Fanuc TP program (LS listing): PNS0002.LS

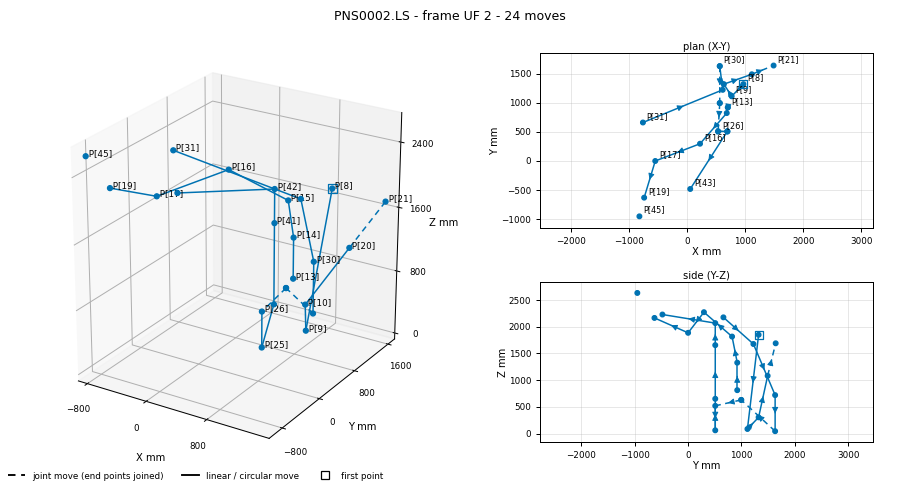
[picture p0: tool path of PNS0002.LS in frame UF 2, 24 of 53 moves have a stored position in this frame; points joined in program order, loops and branches not executed]
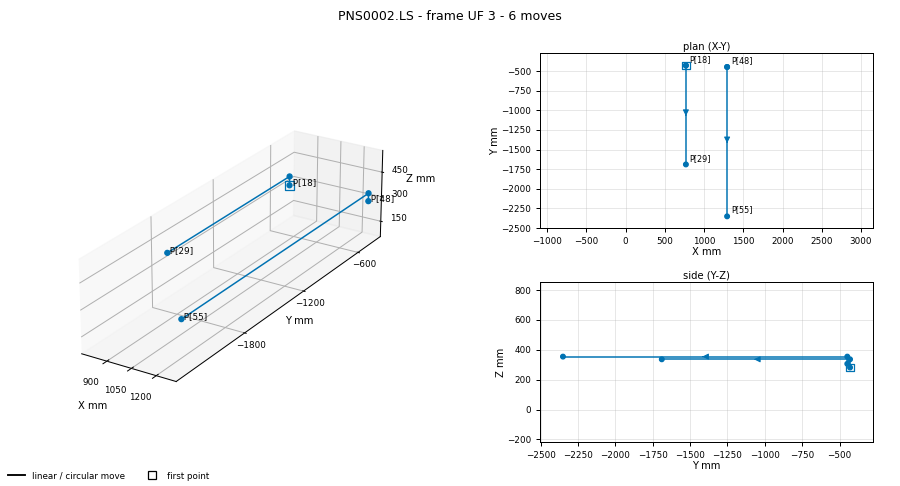
[picture p1: tool path of PNS0002.LS in frame UF 3, 6 of 53 moves have a stored position in this frame; points joined in program order, loops and branches not executed]
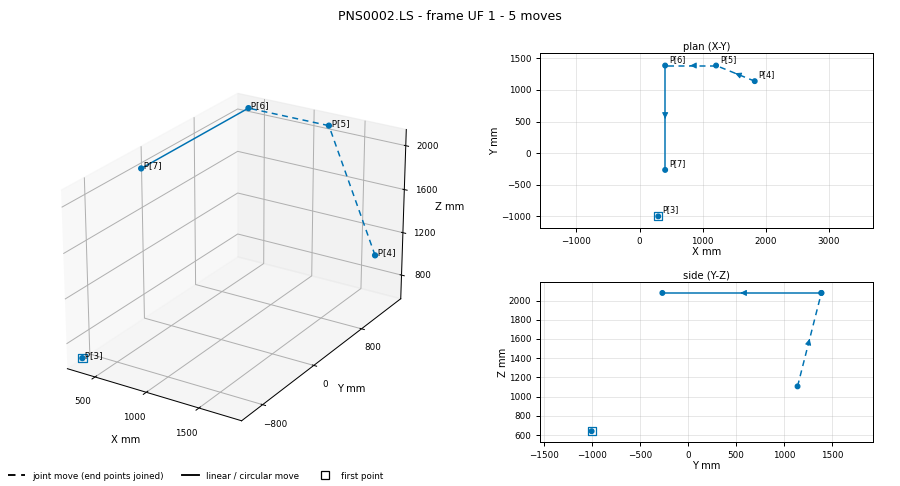
[picture p2: tool path of PNS0002.LS in frame UF 1, 5 of 53 moves have a stored position in this frame; points joined in program order, loops and branches not executed]
/PROG  PNS0002
/ATTR
OWNER		= MNEDITOR;
COMMENT		= "6410816256";
PROG_SIZE	= 5179;
CREATE		= DATE 26-03-31  TIME 11:21:30;
MODIFIED	= DATE 08-10-08  TIME 01:42:36;
FILE_NAME	= ;
VERSION		= 0;
LINE_COUNT	= 173;
MEMORY_SIZE	= 5531;
PROTECT		= READ_WRITE;
STORAGE		= CMOS;
TCD:  STACK_SIZE	= 0,
      TASK_PRIORITY	= 50,
      TIME_SLICE	= 0,
      BUSY_LAMP_OFF	= 0,
      ABORT_REQUEST	= 0,
      PAUSE_REQUEST	= 0;
DEFAULT_GROUP	= 1,*,*,*,*;
CONTROL_CODE	= 00000000 00000000;
/MN
   1:  !6410816256 ;
   2:  !--- INITIALIZE --- ;
   3:  UFRAME_NUM=0 ;
   4:  UTOOL_NUM=1 ;
   5:   ;
   6:J PR[1:HOME] 100% CNT50    ;
   7:   ;
   8:   ;
   9:   ;
  10:  !--- PICK --- ;
  11:  UFRAME_NUM=1 ;
  12:  UTOOL_NUM=1 ;
  13:  TIMER[1]=RESET ;
  14:  TIMER[1]=START ;
  15:   ;
  16:J P[3:INTMPT] 100% CNT10    ;
  17:L P[1:IN FRONT OF IF] 2000mm/sec CNT10    ;
  18:L P[2:ROTATE OVER PICK] 2000mm/sec CNT10    ;
  19:   ;
  20:  !INSERT PART PR ;
  21:  PR[2,3:OFFSET]=400    ;
  22:   ;
  23:L PR[51] 2000mm/sec FINE Offset,PR[2:OFFSET]    ;
  24:L PR[51] 700mm/sec FINE    ;
  25:   ;
  26:  CALL ALL_VAC_ON    ;
  27:   ;
  28:  WAIT   1.00(sec) ;
  29:   ;
  30:L PR[51] 700mm/sec FINE Offset,PR[2:OFFSET]    ;
  31:   ;
  32:J P[4:INTMPT] 100% CNT100    ;
  33:J P[5:INTMPT] 100% CNT100    ;
  34:J P[6:INTMPT] 100% CNT100    ;
  35:L P[7:INTMPT] 2000mm/sec CNT100    ;
  36:   ;
  37:  !--- ZERO TABLE --- ;
  38:  UFRAME_NUM=2 ;
  39:   ;
  40:L P[8:ABOVE ZERO] 1500mm/sec FINE    ;
  41:L P[9:ON ZERO] 1200mm/sec FINE    ;
  42:   ;
  43:  CALL ALL_VAC_OFF    ;
  44:   ;
  45:  !RE-PICK ;
  46:L P[10] 1500mm/sec FINE    ;
  47:L P[20] 1500mm/sec CNT100    ;
  48:J P[21:ROTATE 1] 75% CNT100    ;
  49:J P[22:ROTATE 2] 75% CNT100    ;
  50:J P[11] 75% CNT100    ;
  51:L P[12] 100mm/sec FINE    ;
  52:   ;
  53:  CALL ALL_VAC_ON    ;
  54:   ;
  55:  WAIT   1.00(sec) ;
  56:   ;
  57:L P[11] 155mm/sec FINE    ;
  58:   ;
  59:  !MOVE TO PRESS BREAK ;
  60:L P[13] 2000mm/sec CNT100    ;
  61:L P[14] 1500mm/sec CNT100    ;
  62:L P[15] 1500mm/sec CNT100    ;
  63:L P[16] 1500mm/sec CNT100    ;
  64:L P[17] 1500mm/sec CNT100    ;
  65:   ;
  66:L P[19:STAGED FOR BEND] 500mm/sec FINE    ;
  67:   ;
  68:  !--- BEND 1 --- ;
  69:  UFRAME_NUM=3 ;
  70:   ;
  71:L P[18:INSERT] 500mm/sec FINE    ;
  72:   ;
  73:  CALL PINCH    ;
  74:   ;
  75:  WAIT    .75(sec) ;
  76:   ;
  77:  CALL ALL_VAC_OFF    ;
  78:   ;
  79:  WAIT    .50(sec) ;
  80:   ;
  81:  CALL BEND    ;
  82:   ;
  83:  WAIT   1.00(sec) ;
  84:   ;
  85:  CALL ALL_VAC_ON    ;
  86:   ;
  87:  WAIT   1.00(sec) ;
  88:   ;
  89:  !OUT OF PRESS BREAK ;
  90:L P[28] 700mm/sec FINE    ;
  91:L P[29] 1200mm/sec CNT100    ;
  92:   ;
  93:  !--- ZERO TABLE --- ;
  94:  UFRAME_NUM=2 ;
  95:   ;
  96:  !MOVE TO ZERO ;
  97:L P[31] 1500mm/sec CNT100    ;
  98:L P[32] 1500mm/sec CNT100    ;
  99:L P[30] 1500mm/sec CNT100    ;
 100:L P[33] 500mm/sec FINE    ;
 101:   ;
 102:  CALL ALL_VAC_OFF    ;
 103:   ;
 104:  !REPOS FOR BEND 2 ;
 105:J P[23] 100% CNT100    ;
 106:   ;
 107:J P[24:ZERO J6] 100% CNT100    ;
 108:   ;
 109:J P[26] 100% CNT100    ;
 110:L P[25] 500mm/sec FINE    ;
 111:   ;
 112:L P[27] 1500mm/sec FINE    ;
 113:   ;
 114:  CALL ALL_VAC_ON    ;
 115:   ;
 116:  WAIT   1.00(sec) ;
 117:   ;
 118:  !MOVE TO PRESS BREAK ;
 119:L P[41] 500mm/sec CNT100    ;
 120:L P[42] 1200mm/sec CNT100    ;
 121:L P[43] 1200mm/sec CNT100    ;
 122:L P[44] 1200mm/sec CNT100    ;
 123:L P[45] 1500mm/sec CNT100    ;
 124:   ;
 125:  !--- BEND 2 --- ;
 126:  UFRAME_NUM=3 ;
 127:   ;
 128:L P[48] 500mm/sec FINE    ;
 129:   ;
 130:  CALL PINCH    ;
 131:   ;
 132:  WAIT    .75(sec) ;
 133:   ;
 134:  CALL ALL_VAC_OFF    ;
 135:   ;
 136:  WAIT    .50(sec) ;
 137:   ;
 138:  CALL BEND    ;
 139:   ;
 140:  WAIT   1.00(sec) ;
 141:   ;
 142:  CALL ALL_VAC_ON    ;
 143:   ;
 144:  WAIT   1.00(sec) ;
 145:   ;
 146:  !OUT OF INFEED ;
 147:L P[54] 500mm/sec CNT100    ;
 148:L P[55] 1200mm/sec CNT100    ;
 149:   ;
 150:  !--- OUTFEED --- ;
 151:  UFRAME_NUM=4 ;
 152:   ;
 153:L P[56] 1200mm/sec CNT100    ;
 154:L P[57] 1200mm/sec CNT100    ;
 155:L P[58] 1500mm/sec CNT100    ;
 156:L P[59] 1500mm/sec FINE Offset,PR[2:OFFSET]    ;
 157:L P[59] 500mm/sec FINE    ;
 158:   ;
 159:  CALL ALL_VAC_OFF    ;
 160:   ;
 161:L P[59] 1200mm/sec FINE Offset,PR[2:OFFSET]    ;
 162:   ;
 163:J PR[1:HOME] 100% CNT100    ;
 164:   ;
 165:  TIMER[1]=STOP ;
 166:  R[20]=(TIMER[1]) ;
 167:  !MOVE TO ZERO TABLE ;
 168:  !RE-PICK ;
 169:  !MOVE TO BREAK ;
 170:  !BREAK 1 ;
 171:  !BREAK 2 ;
 172:  !OUTFEED DROP ;
 173:  !HOME ;
/POS
P[1:"IN FRONT OF IF"]{
   GP1:
	UF : 0, UT : 1,		CONFIG : 'N U T, 0, 0, 0',
	X =  3074.267  mm,	Y =      .000  mm,	Z =  -312.592  mm,
	W =   180.000 deg,	P =     -.000 deg,	R =     -.000 deg,
	E1=  1548.896  mm
};
P[2:"ROTATE OVER PICK"]{
   GP1:
	UF : 0, UT : 1,		CONFIG : 'N U T, 0, 0, 0',
	X =  3074.267  mm,	Y =  1357.438  mm,	Z =  -312.592  mm,
	W =   180.000 deg,	P =      .000 deg,	R =    90.000 deg,
	E1=  2600.652  mm
};
P[3:"INTMPT"]{
   GP1:
	UF : 1, UT : 1,		CONFIG : 'N U T, 0, 0, 0',
	X =   295.983  mm,	Y = -1001.060  mm,	Z =   641.268  mm,
	W =   180.000 deg,	P =     -.000 deg,	R =     -.000 deg,
	E1=   633.339  mm
};
P[4:"INTMPT"]{
   GP1:
	UF : 1, UT : 1,		CONFIG : 'N U T, 0, 0, 0',
	X =  1823.555  mm,	Y =  1139.742  mm,	Z =  1107.202  mm,
	W =   180.000 deg,	P =   -40.393 deg,	R =    90.000 deg,
	E1=  2600.652  mm
};
P[5:"INTMPT"]{
   GP1:
	UF : 1, UT : 1,		CONFIG : 'N U T, 0, 0, 0',
	X =  1211.540  mm,	Y =  1387.428  mm,	Z =  2078.739  mm,
	W =   -90.000 deg,	P =   -90.000 deg,	R =     0.000 deg,
	E1=  2600.652  mm
};
P[6:"INTMPT"]{
   GP1:
	UF : 1, UT : 1,		CONFIG : 'N U T, 0, -1, 1',
	X =   405.131  mm,	Y =  1387.428  mm,	Z =  2078.739  mm,
	W =  -111.305 deg,	P =   -90.000 deg,	R =     0.000 deg,
	E1=  1672.415  mm
};
P[7:"INTMPT"]{
   GP1:
	UF : 1, UT : 1,		CONFIG : 'N U T, 0, -1, 1',
	X =   405.131  mm,	Y =  -265.705  mm,	Z =  2078.738  mm,
	W =  -162.943 deg,	P =   -90.000 deg,	R =     0.000 deg,
	E1=  1243.168  mm
};
P[8:"ABOVE ZERO"]{
   GP1:
	UF : 2, UT : 1,		CONFIG : 'N U T, 0, -1, 1',
	X =   970.105  mm,	Y =  1320.827  mm,	Z =  1850.509  mm,
	W =  -179.999 deg,	P =      .001 deg,	R =      .000 deg,
	E1=  2140.441  mm
};
P[9:"ON ZERO"]{
   GP1:
	UF : 2, UT : 1,		CONFIG : 'N U T, 0, -1, 1',
	X =   769.156  mm,	Y =  1111.796  mm,	Z =    85.489  mm,
	W =  -179.997 deg,	P =      .005 deg,	R =     -.999 deg,
	E1=  2580.816  mm
};
P[10:""]{
   GP1:
	UF : 2, UT : 1,		CONFIG : 'N U T, 0, -1, 1',
	X =   635.159  mm,	Y =  1320.793  mm,	Z =   303.508  mm,
	W =  -179.998 deg,	P =      .003 deg,	R =      .000 deg,
	E1=  2580.816  mm
};
P[11:""]{
   GP1:
	UF : 2, UT : 1,
	J1=    18.263 deg,	J2=     6.836 deg,	J3=    -5.826 deg,
	J4=    40.003 deg,	J5=   -26.642 deg,	J6=   234.609 deg,
	E1=  2580.816  mm
};
P[12:""]{
   GP1:
	UF : 2, UT : 1,
	J1=    15.187 deg,	J2=    25.137 deg,	J3=    -9.019 deg,
	J4=    39.754 deg,	J5=   -22.236 deg,	J6=   235.320 deg,
	E1=  2580.816  mm
};
P[13]{
   GP1:
	UF : 2, UT : 1,		CONFIG : 'N U T, 0, -1, 1',
	X =   702.535  mm,	Y =   920.780  mm,	Z =   812.300  mm,
	W =  -179.997 deg,	P =      .004 deg,	R =      .000 deg,
	E1=  2580.816  mm
};
P[14]{
   GP1:
	UF : 2, UT : 1,		CONFIG : 'N U T, 0, 0, 0',
	X =   702.534  mm,	Y =   920.780  mm,	Z =  1327.631  mm,
	W =  -179.997 deg,	P =      .004 deg,	R =      .000 deg,
	E1=  2221.229  mm
};
P[15]{
   GP1:
	UF : 2, UT : 1,		CONFIG : 'N U T, 0, 0, 0',
	X =   684.474  mm,	Y =   823.810  mm,	Z =  1816.677  mm,
	W =   151.491 deg,	P =      .004 deg,	R =     -.001 deg,
	E1=  2195.893  mm
};
P[16]{
   GP1:
	UF : 2, UT : 1,		CONFIG : 'N U T, 0, 0, 1',
	X =   225.090  mm,	Y =   296.601  mm,	Z =  2273.432  mm,
	W =   117.226 deg,	P =    -8.632 deg,	R =   -56.480 deg,
	E1=  1531.414  mm
};
P[17]{
   GP1:
	UF : 2, UT : 1,		CONFIG : 'N U T, 0, 0, 1',
	X =  -544.627  mm,	Y =     -.012  mm,	Z =  1887.026  mm,
	W =   115.203 deg,	P =    -5.023 deg,	R =   -71.293 deg,
	E1=  1531.414  mm
};
P[18:"INSERT"]{
   GP1:
	UF : 3, UT : 1,		CONFIG : 'N U T, 0, 0, 1',
	X =   768.989  mm,	Y =  -429.838  mm,	Z =   281.553  mm,
	W =   179.997 deg,	P =      .001 deg,	R =    82.792 deg,
	E1=  1531.414  mm
};
P[19:"STAGED FOR BEND"]{
   GP1:
	UF : 2, UT : 1,		CONFIG : 'N U T, 0, 0, 1',
	X =  -735.183  mm,	Y =  -630.306  mm,	Z =  2165.855  mm,
	W =   115.200 deg,	P =    -5.019 deg,	R =   -71.293 deg,
	E1=  1531.414  mm
};
P[20:""]{
   GP1:
	UF : 2, UT : 1,		CONFIG : 'N U T, 0, 0, 0',
	X =  1115.243  mm,	Y =  1490.483  mm,	Z =  1081.681  mm,
	W =  -179.996 deg,	P =      .005 deg,	R =      .000 deg,
	E1=  2580.816  mm
};
P[21:"ROTATE 1"]{
   GP1:
	UF : 2, UT : 1,		CONFIG : 'N U T, 0, 0, 1',
	X =  1489.475  mm,	Y =  1640.859  mm,	Z =  1690.573  mm,
	W =    62.575 deg,	P =    32.103 deg,	R =    96.480 deg,
	E1=  2580.816  mm
};
P[22:"ROTATE 2"]{
   GP1:
	UF : 2, UT : 1,
	J1=    15.173 deg,	J2=      .968 deg,	J3=    30.164 deg,
	J4=     9.908 deg,	J5=   -57.573 deg,	J6=   321.680 deg,
	E1=  2580.816  mm
};
P[23]{
   GP1:
	UF : 2, UT : 1,		CONFIG : 'N U T, 0, 0, 1',
	X =   564.202  mm,	Y =   995.409  mm,	Z =   629.737  mm,
	W =   179.952 deg,	P =     1.208 deg,	R =    -2.213 deg,
	E1=  2610.155  mm
};
P[24:"ZERO J6"]{
   GP1:
	UF : 2, UT : 1,		CONFIG : 'N U T, 0, 0, 0',
	X =   564.210  mm,	Y =   995.404  mm,	Z =   629.737  mm,
	W =   179.930 deg,	P =     1.207 deg,	R =    46.747 deg,
	E1=  2610.155  mm
};
P[25]{
   GP1:
	UF : 2, UT : 1,		CONFIG : 'N U T, 0, 0, 0',
	X =   535.405  mm,	Y =   508.764  mm,	Z =    59.990  mm,
	W =  -176.805 deg,	P =      .463 deg,	R =    46.253 deg,
	E1=  2610.155  mm
};
P[26]{
   GP1:
	UF : 2, UT : 1,		CONFIG : 'N U T, 0, 0, 0',
	X =   535.407  mm,	Y =   508.762  mm,	Z =   518.988  mm,
	W =  -176.805 deg,	P =      .463 deg,	R =    46.252 deg,
	E1=  2610.155  mm
};
P[27]{
   GP1:
	UF : 2, UT : 1,		CONFIG : 'N U T, 0, 0, 0',
	X =   694.414  mm,	Y =   508.757  mm,	Z =   650.986  mm,
	W =  -176.803 deg,	P =      .462 deg,	R =    46.252 deg,
	E1=  2610.155  mm
};
P[28:""]{
   GP1:
	UF : 3, UT : 1,		CONFIG : 'N U T, 0, 0, 1',
	X =   768.987  mm,	Y =  -429.847  mm,	Z =   336.553  mm,
	W =   179.997 deg,	P =      .001 deg,	R =    82.792 deg,
	E1=  1531.414  mm
};
P[29:""]{
   GP1:
	UF : 3, UT : 1,		CONFIG : 'N U T, 0, 0, 1',
	X =   768.987  mm,	Y = -1689.847  mm,	Z =   336.553  mm,
	W =   179.997 deg,	P =      .001 deg,	R =    82.792 deg,
	E1=   885.138  mm
};
P[30]{
   GP1:
	UF : 2, UT : 1,		CONFIG : 'N U T, 0, 0, 1',
	X =   564.157  mm,	Y =  1630.434  mm,	Z =   719.716  mm,
	W =   179.951 deg,	P =     1.205 deg,	R =   -43.213 deg,
	E1=  2610.155  mm
};
P[31]{
   GP1:
	UF : 2, UT : 1,		CONFIG : 'N U T, 0, 0, 1',
	X =  -756.542  mm,	Y =   661.571  mm,	Z =  2176.748  mm,
	W =   153.444 deg,	P =    26.651 deg,	R =   -28.332 deg,
	E1=   650.447  mm
};
P[32]{
   GP1:
	UF : 2, UT : 1,		CONFIG : 'N U T, 0, 0, 1',
	X =   615.016  mm,	Y =  1223.310  mm,	Z =  1677.627  mm,
	W =  -179.363 deg,	P =      .470 deg,	R =   -43.202 deg,
	E1=  1757.984  mm
};
P[33:""]{
   GP1:
	UF : 2, UT : 1,		CONFIG : 'N U T, 0, 0, 1',
	X =   564.153  mm,	Y =  1630.436  mm,	Z =    43.712  mm,
	W =   179.952 deg,	P =     1.204 deg,	R =   -43.213 deg,
	E1=  2610.155  mm
};
P[41]{
   GP1:
	UF : 2, UT : 1,		CONFIG : 'N U T, 0, 0, 0',
	X =   694.433  mm,	Y =   508.743  mm,	Z =  1655.979  mm,
	W =  -176.803 deg,	P =      .462 deg,	R =    46.253 deg,
	E1=  2049.709  mm
};
P[42]{
   GP1:
	UF : 2, UT : 1,		CONFIG : 'N U T, 0, 0, 0',
	X =   694.503  mm,	Y =   508.695  mm,	Z =  2068.966  mm,
	W =   159.538 deg,	P =    37.933 deg,	R =     -.769 deg,
	E1=  2049.709  mm
};
P[43]{
   GP1:
	UF : 2, UT : 1,		CONFIG : 'N U T, 0, 0, 0',
	X =    56.692  mm,	Y =  -481.063  mm,	Z =  2229.808  mm,
	W =   124.382 deg,	P =    41.784 deg,	R =   -28.741 deg,
	E1=  1111.976  mm
};
P[44]{
   GP1:
	UF : 2, UT : 1,
	J1=   -22.722 deg,	J2=   -12.962 deg,	J3=    -6.975 deg,
	J4=     -.000 deg,	J5=   -83.025 deg,	J6=   -62.136 deg,
	E1=   801.510  mm
};
P[45]{
   GP1:
	UF : 2, UT : 1,		CONFIG : 'N U T, 0, 0, 0',
	X =  -816.862  mm,	Y =  -951.537  mm,	Z =  2634.093  mm,
	W =   115.571 deg,	P =    10.679 deg,	R =   -63.868 deg,
	E1=   801.510  mm
};
P[48]{
   GP1:
	UF : 3, UT : 1,		CONFIG : 'N U T, 0, 0, 0',
	X =  1293.952  mm,	Y =  -448.177  mm,	Z =   306.614  mm,
	W =   179.998 deg,	P =      .002 deg,	R =   100.145 deg,
	E1=   801.510  mm
};
P[54]{
   GP1:
	UF : 3, UT : 1,		CONFIG : 'N U T, 0, 0, 0',
	X =  1293.952  mm,	Y =  -448.177  mm,	Z =   354.614  mm,
	W =   179.998 deg,	P =      .002 deg,	R =   100.145 deg,
	E1=   795.174  mm
};
P[55]{
   GP1:
	UF : 3, UT : 1,		CONFIG : 'N U T, 0, 0, 0',
	X =  1293.952  mm,	Y = -2351.177  mm,	Z =   354.614  mm,
	W =   179.998 deg,	P =      .002 deg,	R =   100.145 deg,
	E1=    91.875  mm
};
P[56]{
   GP1:
	UF : 4, UT : 1,		CONFIG : 'N U T, 0, 0, 0',
	X =  2909.047  mm,	Y = -1041.823  mm,	Z =   935.614  mm,
	W =   166.201 deg,	P =   -50.073 deg,	R =   -13.412 deg,
	E1=    91.875  mm
};
P[57]{
   GP1:
	UF : 4, UT : 1,		CONFIG : 'N U T, 0, 0, 0',
	X =  2832.047  mm,	Y =  -301.823  mm,	Z =   935.614  mm,
	W =  -180.000 deg,	P =     -.000 deg,	R =   -43.000 deg,
	E1=    91.875  mm
};
P[58]{
   GP1:
	UF : 4, UT : 1,		CONFIG : 'N U T, 0, 0, 0',
	X =  2061.047  mm,	Y =   979.177  mm,	Z =   359.614  mm,
	W =   180.000 deg,	P =     -.000 deg,	R =   -43.000 deg,
	E1=    91.875  mm
};
P[59]{
   GP1:
	UF : 4, UT : 1,		CONFIG : 'N U T, 0, 0, 0',
	X =  1570.047  mm,	Y =   944.177  mm,	Z =     9.614  mm,
	W =   180.000 deg,	P =      .000 deg,	R =   -43.000 deg,
	E1=    91.875  mm
};
/END
